VISUALIZATION Run  // 1280x800, background image BackGroundImagePool_SVG.Background_Sides
END_VISUALIZATION

(* stored: Version 1.1.0.1, ProductVersion 3.1.4024.5
   Visu Run: Id {49da977c-55e0-4e44-8992-2a040fff7bb6} *)
